{attribute 'qualified_only'}
{attribute 'strict'}
{attribute 'to_string'}
TYPE E_3002_Set_ESTOP :
(
	Release_ESTOP := 0,
	Set_ESTOP:=1
)UINT;
END_TYPE

(* stored: Version 1.1.0.1, ProductVersion 3.1.4026.17
   DUT E_3002_Set_ESTOP: Id {afa45918-f8ba-4668-a840-34d3ce59e676} *)
